{attribute 'GeneratedUsingTerminal: EK1122-0000-0018'}
{attribute addProperty BoxType "EK1122-0000-0018"}
{attribute addProperty Id "Beckhoff_EP8xxxsub_EK1100EK1100_AB5A94672A_0001_EP8309_0022_0021EP8309_35A864DD70A_0002_EP8309_1022_0016EP8309_35A864DD70A_0003_EP8309_1022_0017EP8309_35A864DD70A_0004_EP8309_1022_0018EP8309_35A864DD70"}
{attribute addProperty CRC "1487746608"}
{attribute addProperty Size "282"}
TYPE Beckhoff_EP8xxxEK1122_58AD3630 EXTENDS EK1122_AB5A9467 :
STRUCT
	{attribute addProperty Name "Beckhoff_EP8xxxsub_EK1100"}
	Beckhoff_EP8xxxsub_EK1100 : EK1100_AB5A9467;
	{attribute addProperty Name "A_0001_EP8309_0022_0021"}
	A_0001_EP8309_0022_0021 : EP8309_35A864DD;
	{attribute addProperty Name "A_0002_EP8309_1022_0016"}
	A_0002_EP8309_1022_0016 : EP8309_35A864DD;
	{attribute addProperty Name "A_0003_EP8309_1022_0017"}
	A_0003_EP8309_1022_0017 : EP8309_35A864DD;
	{attribute addProperty Name "A_0004_EP8309_1022_0018"}
	A_0004_EP8309_1022_0018 : EP8309_35A864DD;
END_STRUCT
END_TYPE

(* stored: Version 1.2.0.0, ProductVersion 3.1.4024.9
   DUT Beckhoff_EP8xxxEK1122_58AD3630: Id {b147612d-d9b6-4a9e-8689-37082f8d5b1b} *)
